TYPE ST_SolventInfo :
STRUCT
    sName     : STRING(50); // Name of the solvent (e.g., Water, Methanol)
    iRevision : INT; // Revision/version of the solvent definition
END_STRUCT
END_TYPE

(* stored: Version 1.1.0.1, ProductVersion 3.1.4024.12
   DUT ST_SolventInfo: Id {036b89d2-a065-43bf-a66c-f961e1294041} *)
